// TIA Portal V17 export
// export: Created 2023-04-03T06:31:41.7365661Z, ExportSetting WithDefaults, DisplayName Totally Integrated Automation Portal, DisplayVersion V17 Update 4, DisplayName TIA Portal Openness, DisplayVersion V17 Update 4, DisplayName TIA Portal Version Control Interface, DisplayVersion V17, DisplayName STEP 7 Professional, DisplayVersion V17 Update 4, DisplayName STEP 7 Safety, DisplayVersion V17, DisplayName WinCC Professional, DisplayVersion V17 Update 4
TYPE "CATL_CELL_T"
// stored: IsFailsafeCompliant false
   STRUCT
      CSC1_Temp_Cell1 : Real;
      CSC1_Temp_Cell2 : Real;
      CSC1_Temp_Cell3 : Real;
      CSC1_Temp_Cell4 : Real;
      CSC1_Temp_Cell5 : Real;
      CSC1_Temp_Cell6 : Real;
      CSC1_Temp_Cell7 : Real;
      CSC1_Temp_Cell8 : Real;
      CSC2_Temp_Cell1 : Real;
      CSC2_Temp_Cell2 : Real;
      CSC2_Temp_Cell3 : Real;
      CSC2_Temp_Cell4 : Real;
      CSC2_Temp_Cell5 : Real;
      CSC2_Temp_Cell6 : Real;
      CSC2_Temp_Cell7 : Real;
      CSC2_Temp_Cell8 : Real;
      CSC3_Temp_Cell1 : Real;
      CSC3_Temp_Cell2 : Real;
      CSC3_Temp_Cell3 : Real;
      CSC3_Temp_Cell4 : Real;
      CSC3_Temp_Cell5 : Real;
      CSC3_Temp_Cell6 : Real;
      CSC3_Temp_Cell7 : Real;
      CSC3_Temp_Cell8 : Real;
      CSC4_Temp_Cell1 : Real;
      CSC4_Temp_Cell2 : Real;
      CSC4_Temp_Cell3 : Real;
      CSC4_Temp_Cell4 : Real;
      CSC4_Temp_Cell5 : Real;
      CSC4_Temp_Cell6 : Real;
      CSC4_Temp_Cell7 : Real;
      CSC4_Temp_Cell8 : Real;
      CSC5_Temp_Cell1 : Real;
      CSC5_Temp_Cell2 : Real;
      CSC5_Temp_Cell3 : Real;
      CSC5_Temp_Cell4 : Real;
      CSC5_Temp_Cell5 : Real;
      CSC5_Temp_Cell6 : Real;
      CSC5_Temp_Cell7 : Real;
      CSC5_Temp_Cell8 : Real;
      CSC6_Temp_Cell1 : Real;
      CSC6_Temp_Cell2 : Real;
      CSC6_Temp_Cell3 : Real;
      CSC6_Temp_Cell4 : Real;
      CSC6_Temp_Cell5 : Real;
      CSC6_Temp_Cell6 : Real;
      CSC6_Temp_Cell7 : Real;
      CSC6_Temp_Cell8 : Real;
      CSC7_Temp_Cell1 : Real;
      CSC7_Temp_Cell2 : Real;
      CSC7_Temp_Cell3 : Real;
      CSC7_Temp_Cell4 : Real;
      CSC7_Temp_Cell5 : Real;
      CSC7_Temp_Cell6 : Real;
      CSC7_Temp_Cell7 : Real;
      CSC7_Temp_Cell8 : Real;
      CSC8_Temp_Cell1 : Real;
      CSC8_Temp_Cell2 : Real;
      CSC8_Temp_Cell3 : Real;
      CSC8_Temp_Cell4 : Real;
      CSC8_Temp_Cell5 : Real;
      CSC8_Temp_Cell6 : Real;
      CSC8_Temp_Cell7 : Real;
      CSC8_Temp_Cell8 : Real;
   END_STRUCT;
END_TYPE
